(* CODESYS project Progetto_RECOVERED_2026-03-03T14-50-17.project

Project tree, tasks and I/O mapping:
  Device : CODESYS Control Win V3 x64, CODESYS, version 3.5.21.30
    application Application
      libraries: Standard, 3.5.18.0 (System)
      task MainTask (cyclic, interval t#20ms, priority 1) calls PLC_PRG, Controller
      program PLC_PRG [SFC]: END_MOVINGX1, END_MOVINGX, MOVE_X_SX, Trasporting_dx_entry, PickPlace_sx_active, MOVE_SX, Return_dx_active, MOVE_Z_SX, Loading_active, Place_sx_exit, Trasporting_dx_active, High_dx_exit, Start_active
      global variables FIO
      program Controller [FBD]
      Symbols
*)

// Device/Application/FIO
{attribute 'qualified_only'}
VAR_GLOBAL
	
	//pulsanti 
	IN_START: BOOL;
	IN_STOP: BOOL;
	IN_RESET: BOOL;
	IN_EMERGENCYSTOP: BOOL;
	
	//----SMISTAMENTO---
	//SENSORS
	IN_HIGHSEN: BOOL; //sensore pacchi alti
	IN_LOWSEN: BOOL; //sensore pacchi bassi
	
	IN_PSEN: BOOL; //sensore pallet = ingresso al transger
	IN_LOADED: BOOL; //sensore "pacco caricato" sul transfer
	
	IN_LENTRY: BOOL; //sensore ingresso nastro sx
	IN_LEXIT: BOOL; //sensore uscita nastro sx
	IN_RENTRY: BOOL; //sensore ingresso nastro dx
	IN_REXIT: BOOL; //sensore uscita nastro dx
	
	// ACTUATORS
	OUT_CONVENTRY: BOOL; //nastro d'ingresso
	OUT_EMITTER: BOOL;
	
	OUT_LOAD: BOOL; //inserisce il pacco sul transfer
	OUT_UNLOAD: BOOL; //rimuove il pacco dal transfer
	
	OUT_LTRANS: BOOL; //muove a sinistra il pacco
	OUT_RTRANS: BOOL; //attiva il transfer per muovere a destra il pacco
	
	OUT_CONVLEFT: BOOL; //nastro uscita sx
	OUT_CONVRIGHT: BOOL; //nastro uscita dx
	
	OUT_STARTLIGHT: BOOL;
	OUT_STOPLIGHT: BOOL;
	OUT_RESETLIGHT: BOOL;
	
	//---- WAREHOUSE DX ----
	//SENSORS
	IN_DX_LEFT: BOOL;
	IN_DX_RIGHT: BOOL;
	IN_DX_LOAD: BOOL;
	IN_DX_UNLOAD: BOOL;
	IN_DX_MIDDLE: BOOL;
	IN_DX_MOVING_X: BOOL;
	IN_DX_MOVING_Z: BOOL;
	
	//ACTUATORS
	OUT_DX_LIFT: BOOL;
	OUT_DX_LFORK: BOOL;
	OUT_DX_RFORK: BOOL;
	OUT_DX_LOADCONV: BOOL;
	OUT_DX_UNLOADCONV: BOOL;
	OUT_DX_TARGETPOS: WORD := 0;
	
	//---- Pick Place DX ----
	//SENSORS
	IN_LX_MOVING_Z: BOOL; //azze z in mov
	IN_LX_DETECTED: BOOL; //pezzo detected
	IN_LX_MOVING_X: BOOL; //asse x in mov
	IN_LX_LENTRY2: BOOL; //fine conv pick
	IN_LX_LEXIT2: BOOL; //fine conv place
	
	//ACTUATORS
	OUT_LX_CONVEYOR2: BOOL;
	OUT_LX_GRAB: BOOL;
	OUT_LX_MOVEZ: BOOL; //su giu
	OUT_LX_MOVEX: BOOL; //trasferisce
	
END_VAR

// Device/Application/PLC_PRG
 PROGRAM PLC_PRG
VAR
	IS_HIGH: BOOL;
	
	NEXT_POSITION: WORD := 0;
	F_TRIG_0: F_TRIG;
	F_TRIG_1: F_TRIG;
	
	Timer: TON;
	Timer_transf_sx: TON;
	Timer_grab1: TON;
	Timer_place: TON;
	Timer_goback: TON;
	Timer_movex: TON;
	
	IS_PLACED: BOOL;
	
	Timer_conveyor: TON;
END_VAR
VAR // added by the converter: edge detectors and wires of the graphical bodies
    _ft1 : F_TRIG;
    _w1 : BOOL;
END_VAR

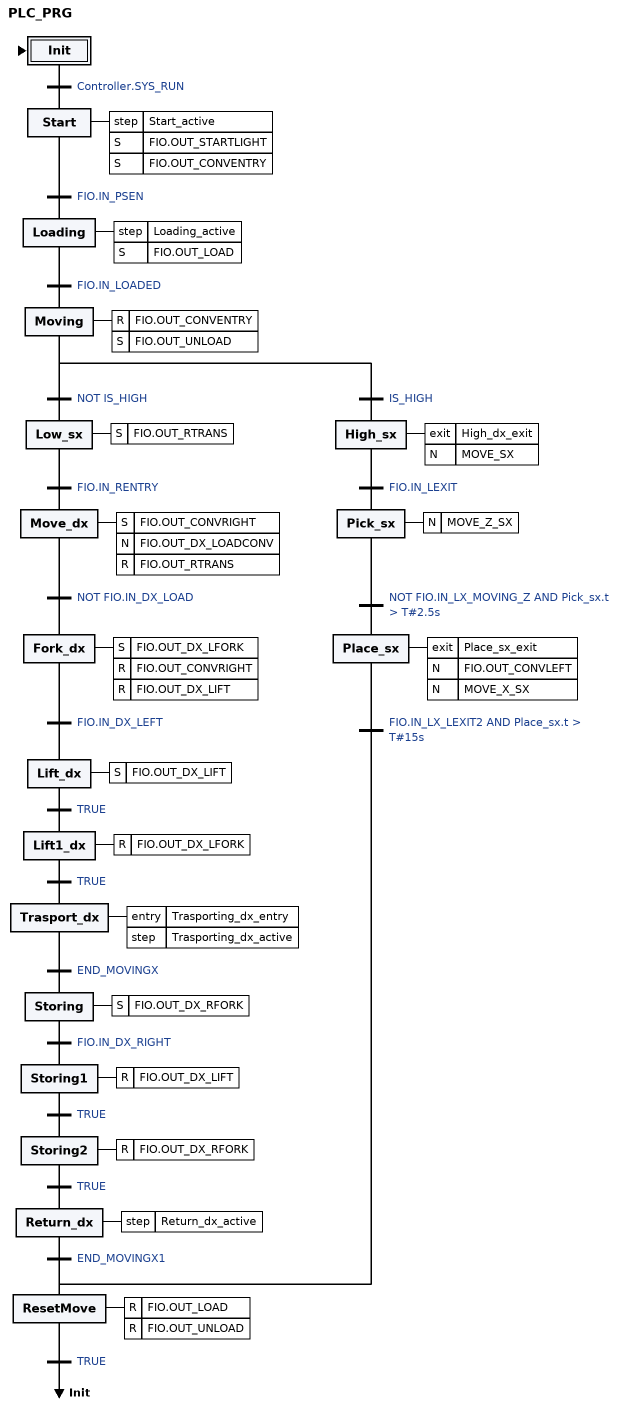
INITIAL_STEP Init:
END_STEP
TRANSITION FROM Init TO Start
    := Controller.SYS_RUN;
END_TRANSITION
STEP Start:  // min time T#1s
    Start_active(N);  // step action
    FIO.OUT_STARTLIGHT(S);
    FIO.OUT_CONVENTRY(S);
END_STEP
TRANSITION FROM Start TO Loading
    := FIO.IN_PSEN;
END_TRANSITION
STEP Loading:
    Loading_active(N);  // step action
    FIO.OUT_LOAD(S);
END_STEP
TRANSITION FROM Loading TO Moving
    := FIO.IN_LOADED;
END_TRANSITION
STEP Moving:  // min time T#2s
    FIO.OUT_CONVENTRY(R);
    FIO.OUT_UNLOAD(S);
END_STEP
TRANSITION FROM Moving TO Low_sx
    := NOT IS_HIGH;
END_TRANSITION
// macro Destra begins
STEP Low_sx:  // min time T#1.5s
    FIO.OUT_RTRANS(S);
END_STEP
TRANSITION FROM Low_sx TO Move_dx
    := FIO.IN_RENTRY;
END_TRANSITION
STEP Move_dx:  // min time T#3s
    FIO.OUT_CONVRIGHT(S);
    FIO.OUT_DX_LOADCONV(N);
    FIO.OUT_RTRANS(R);
END_STEP
TRANSITION FROM Move_dx TO Fork_dx
    := NOT FIO.IN_DX_LOAD;
END_TRANSITION
// macro Receiving_dx begins
STEP Fork_dx:
    FIO.OUT_DX_LFORK(S);
    FIO.OUT_CONVRIGHT(R);
    FIO.OUT_DX_LIFT(R);
END_STEP
TRANSITION FROM Fork_dx TO Lift_dx
    := FIO.IN_DX_LEFT;
END_TRANSITION
STEP Lift_dx:  // min time T#2s
    FIO.OUT_DX_LIFT(S);
END_STEP
TRANSITION FROM Lift_dx TO Lift1_dx
    := TRUE;
END_TRANSITION
STEP Lift1_dx:  // min time T#2.5s
    FIO.OUT_DX_LFORK(R);
END_STEP
TRANSITION FROM Lift1_dx TO Trasport_dx
    := TRUE;
END_TRANSITION
STEP Trasport_dx:
    Trasporting_dx_entry(P1);  // entry action
    Trasporting_dx_active(N);  // step action
END_STEP
TRANSITION FROM Trasport_dx TO Storing
    := END_MOVINGX;
END_TRANSITION
// macro Store_dx begins
STEP Storing:
    FIO.OUT_DX_RFORK(S);
END_STEP
TRANSITION FROM Storing TO Storing1
    := FIO.IN_DX_RIGHT;
END_TRANSITION
STEP Storing1:  // min time T#3s
    FIO.OUT_DX_LIFT(R);
END_STEP
TRANSITION FROM Storing1 TO Storing2
    := TRUE;
END_TRANSITION
STEP Storing2:  // min time T#3s
    FIO.OUT_DX_RFORK(R);
END_STEP
TRANSITION FROM Storing2 TO Return_dx
    := TRUE;
END_TRANSITION
STEP Return_dx:
    Return_dx_active(N);  // step action
END_STEP
TRANSITION FROM Return_dx TO ResetMove
    := END_MOVINGX1;
END_TRANSITION
TRANSITION FROM Moving TO High_sx
    := IS_HIGH;
END_TRANSITION
// macro Sinistra begins
STEP High_sx:  // min time T#1.5s
    High_dx_exit(P0);  // exit action
    MOVE_SX(N);
END_STEP
TRANSITION FROM High_sx TO Pick_sx
    := FIO.IN_LEXIT;
END_TRANSITION
STEP Pick_sx:
    MOVE_Z_SX(N);
END_STEP
TRANSITION FROM Pick_sx TO Place_sx
    := NOT FIO.IN_LX_MOVING_Z AND Pick_sx.t > T#2.5s;
END_TRANSITION
STEP Place_sx:
    Place_sx_exit(P0);  // exit action
    FIO.OUT_CONVLEFT(N);
    MOVE_X_SX(N);
END_STEP
TRANSITION FROM Place_sx TO ResetMove
    := FIO.IN_LX_LEXIT2 AND Place_sx.t > T#15s;
END_TRANSITION
STEP ResetMove:  // min time T#2s
    FIO.OUT_LOAD(R);
    FIO.OUT_UNLOAD(R);
END_STEP
TRANSITION FROM ResetMove TO Init
    := TRUE;
END_TRANSITION

TRANSITION END_MOVINGX1:
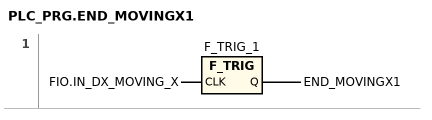
// NETWORK 1
F_TRIG_1(CLK := FIO.IN_DX_MOVING_X); // F_TRIG
END_MOVINGX1 := F_TRIG_1.Q;
END_TRANSITION

TRANSITION END_MOVINGX:
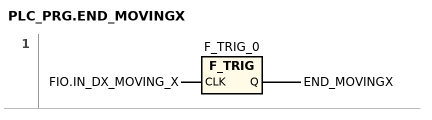
// NETWORK 1
F_TRIG_0(CLK := FIO.IN_DX_MOVING_X); // F_TRIG
END_MOVINGX := F_TRIG_0.Q;
END_TRANSITION

ACTION MOVE_X_SX:
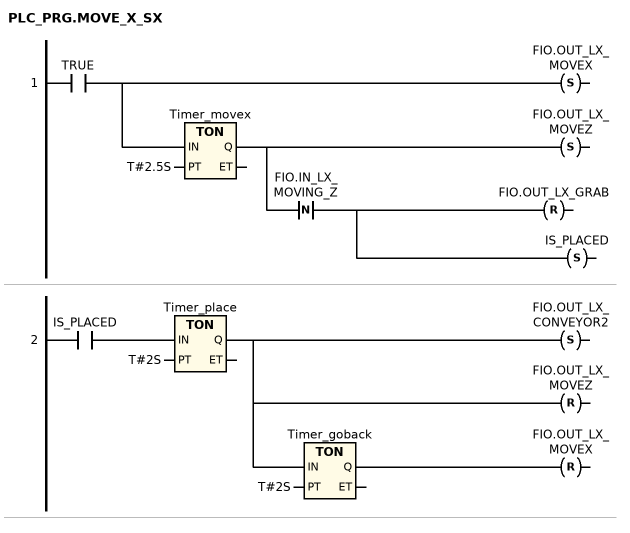
// NETWORK 1
FIO.OUT_LX_MOVEX S= TRUE;
Timer_movex(IN := TRUE, PT := T#2.5S); // TON
FIO.OUT_LX_MOVEZ S= Timer_movex.Q;
_ft1(CLK := FIO.IN_LX_MOVING_Z);
_w1 := Timer_movex.Q AND _ft1.Q;
FIO.OUT_LX_GRAB R= _w1;
IS_PLACED S= _w1;

// NETWORK 2
Timer_place(IN := IS_PLACED, PT := T#2S); // TON
FIO.OUT_LX_CONVEYOR2 S= Timer_place.Q;
FIO.OUT_LX_MOVEZ R= Timer_place.Q;
Timer_goback(IN := Timer_place.Q, PT := T#2S); // TON
FIO.OUT_LX_MOVEX R= Timer_goback.Q;
END_ACTION

ACTION Trasporting_dx_entry:
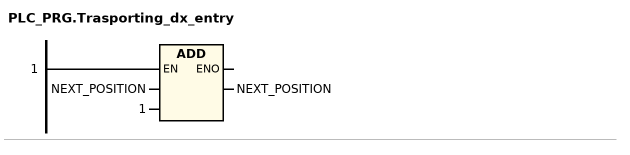
// NETWORK 1
NEXT_POSITION := NEXT_POSITION + 1;
END_ACTION

ACTION PickPlace_sx_active:

END_ACTION

ACTION MOVE_SX:
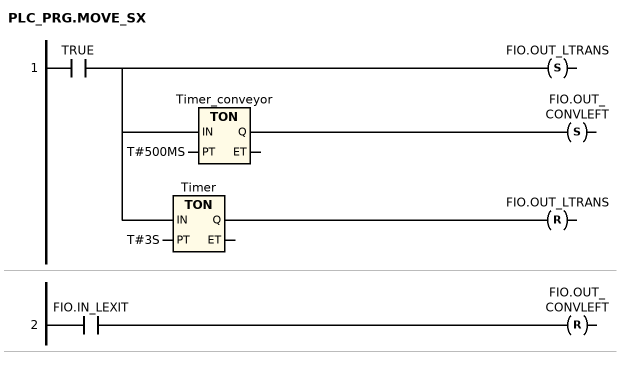
// NETWORK 1
FIO.OUT_LTRANS S= TRUE;
Timer_conveyor(IN := TRUE, PT := T#500MS); // TON
FIO.OUT_CONVLEFT S= Timer_conveyor.Q;
Timer(IN := TRUE, PT := T#3S); // TON
FIO.OUT_LTRANS R= Timer.Q;

// NETWORK 2
FIO.OUT_CONVLEFT R= FIO.IN_LEXIT;
END_ACTION

ACTION Return_dx_active:
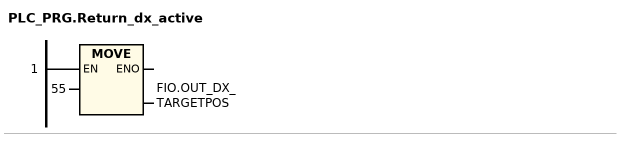
// NETWORK 1
FIO.OUT_DX_TARGETPOS := 55;
END_ACTION

ACTION MOVE_Z_SX:
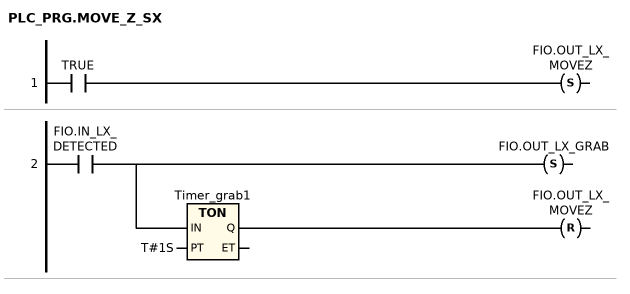
// NETWORK 1
FIO.OUT_LX_MOVEZ S= TRUE;

// NETWORK 2
FIO.OUT_LX_GRAB S= FIO.IN_LX_DETECTED;
Timer_grab1(IN := FIO.IN_LX_DETECTED, PT := T#1S); // TON
FIO.OUT_LX_MOVEZ R= Timer_grab1.Q;
END_ACTION

ACTION Loading_active:
IF FIO.IN_HIGHSEN THEN
    IS_HIGH := TRUE;
END_IF
END_ACTION

ACTION Place_sx_exit:
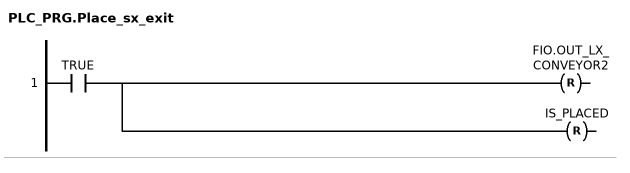
// NETWORK 1
FIO.OUT_LX_CONVEYOR2 R= TRUE;
IS_PLACED R= TRUE;
END_ACTION

ACTION Trasporting_dx_active:
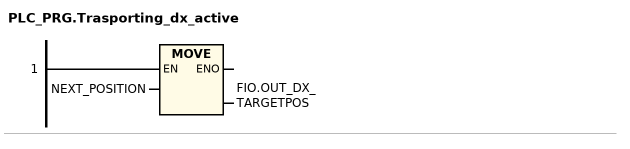
// NETWORK 1
FIO.OUT_DX_TARGETPOS := NEXT_POSITION;
END_ACTION

ACTION High_dx_exit:
IS_HIGH := FALSE;
END_ACTION

ACTION Start_active:

END_ACTION

END_PROGRAM

// Device/Application/Controller
PROGRAM Controller
VAR
	RS_0: RS;
	SYS_RUN: BOOL;
END_VAR

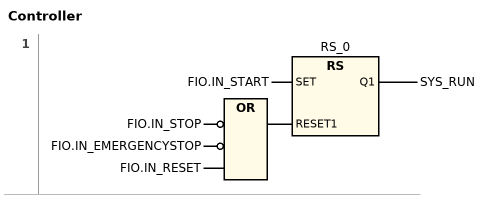
// NETWORK 1
RS_0(SET := FIO.IN_START, RESET1 := NOT FIO.IN_STOP OR NOT FIO.IN_EMERGENCYSTOP OR FIO.IN_RESET); // RS
SYS_RUN := RS_0.Q1;

END_PROGRAM
